(* IEC 61131-3 sources: RL_MAR/experiments/comparison/llm4plc/results/gpt-4o-mini_20260506_100619/20260506_101124, 4 files *)

(* ---- generated_code_iteration_0.st ---- *)
ructured-text
FUNCTION_BLOCK TruckGarage
VAR_INPUT
    enter_flag : BOOL;
    exit_flag : BOOL;
    VehicleNumber_in : INT;
END_VAR
VAR_OUTPUT
    truck : T_TRUCK_INFO;
END_VAR
VAR_IN_OUT
    garage : ARRAY[1..3, 1..5] OF T_GARAGE_SLOT;
END_VAR
VAR
    state : INT; // THE STATE VARIABLE
    row : INT; // THE CURRENT row being checked for parking
    col : INT; // THE CURRENT column being checked for parking
    found : BOOL; // Flag to indicate if a parking space has been found
    exit_row : INT; // Row of the vehicle to be exited
    exit_col : INT; // Column of the vehicle to be exited
    exit_found : BOOL; // Flag to indicate if the vehicle to be exited is found
END_VAR

// STATE MACHINE
IF state = 0 THEN // IDLE STATE
    IF enter_flag = TRUE AND exit_flag = FALSE THEN
        state := 1; // Transition to ALLOCATE PARKING SPACE
    ELSIF exit_flag = TRUE AND enter_flag = FALSE THEN
        state := 2; // Transition to RELEASE PARKING SPACE
    END_IF

ELSIF state = 1 THEN // ALLOCATE PARKING SPACE
    found := FALSE;
    FOR row := 3 TO 1 BY -1 DO
        FOR col := 5 TO 1 BY -1 DO
            IF garage[row, col].Occupied = FALSE THEN
                garage[row, col].Occupied := TRUE;
                garage[row, col].VehicleNumber := VehicleNumber_in;
                truck.row := row;
                truck.col := col;
                truck.VehicleNumber := VehicleNumber_in;
                found := TRUE;
                EXIT; // Exit the inner loop
            END_IF
        END_FOR
        IF found THEN
            EXIT; // Exit the outer loop
        END_IF
    END_FOR
    state := 0; // Transition back to IDLE STATE

ELSIF state = 2 THEN // RELEASE PARKING SPACE
    exit_found := FALSE;
    FOR row := 1 TO 3 DO
        FOR col := 1 TO 5 DO
            IF garage[row, col].VehicleNumber = VehicleNumber_in THEN
                garage[row, col].Occupied := FALSE;
                garage[row, col].VehicleNumber := 0; // Clear the VehicleNumber
                truck.row := row;
                truck.col := col;
                truck.VehicleNumber := VehicleNumber_in;
                exit_found := TRUE;
                EXIT; // Exit the inner loop
            END_IF
        END_FOR
        IF exit_found THEN
            EXIT; // Exit the outer loop
        END_IF
    END_FOR
    state := 0; // Transition back to IDLE STATE
END_IF

END_FUNCTION_BLOCK

(* ---- generated_code_iteration_1.st ---- *)
START_REASON
The errors occurred because the type 'T_TRUCK_INFO' is unknown in the context of the provided Structured Text (ST) code. This suggests that the type definition for 'T_TRUCK_INFO' has not been included or defined in the code. Additionally, the variable sections should be closed with "END_VAR" instead of "END_VAR_OUTPUT" or "END_VAR_INPUT". To resolve these issues, I will define the necessary types and ensure the variable sections are correctly closed.
END_REASON

START_ST
FUNCTION_BLOCK TruckGarage
VAR_INPUT
    enter_flag : BOOL;
    exit_flag : BOOL;
    VehicleNumber_in : INT;
END_VAR
VAR_OUTPUT
    truck : T_TRUCK_INFO;
END_VAR
VAR_IN_OUT
    garage : ARRAY[1..3, 1..5] OF T_GARAGE_SLOT;
END_VAR
VAR
    state : INT; // THE STATE VARIABLE
    row : INT; // THE CURRENT row being checked for parking
    col : INT; // THE CURRENT column being checked for parking
    found : BOOL; // Flag to indicate if a parking space has been found
    exit_row : INT; // Row of the vehicle to be exited
    exit_col : INT; // Column of the vehicle to be exited
    exit_found : BOOL; // Flag to indicate if the vehicle to be exited is found
END_VAR

// TYPE DEFINITIONS
TYPE T_TRUCK_INFO :
STRUCT
    row : INT;
    col : INT;
    VehicleNumber : INT;
END_STRUCT
END_TYPE

TYPE T_GARAGE_SLOT :
STRUCT
    Occupied : BOOL;
    VehicleNumber : INT;
END_STRUCT
END_TYPE

// STATE MACHINE
IF state = 0 THEN // IDLE STATE
    IF enter_flag = TRUE AND exit_flag = FALSE THEN
        state := 1; // Transition to ALLOCATE PARKING SPACE
    ELSIF exit_flag = TRUE AND enter_flag = FALSE THEN
        state := 2; // Transition to RELEASE PARKING SPACE
    END_IF

ELSIF state = 1 THEN // ALLOCATE PARKING SPACE
    found := FALSE;
    FOR row := 3 TO 1 BY -1 DO
        FOR col := 5 TO 1 BY -1 DO
            IF garage[row, col].Occupied = FALSE THEN
                garage[row, col].Occupied := TRUE;
                garage[row, col].VehicleNumber := VehicleNumber_in;
                truck.row := row;
                truck.col := col;
                truck.VehicleNumber := VehicleNumber_in;
                found := TRUE;
                EXIT; // Exit the inner loop
            END_IF
        END_FOR
        IF found THEN
            EXIT; // Exit the outer loop
        END_IF
    END_FOR
    state := 0; // Transition back to IDLE STATE

ELSIF state = 2 THEN // RELEASE PARKING SPACE
    exit_found := FALSE;
    FOR row := 1 TO 3 DO
        FOR col := 1 TO 5 DO
            IF garage[row, col].VehicleNumber = VehicleNumber_in THEN
                garage[row, col].Occupied := FALSE;
                garage[row, col].VehicleNumber := 0; // Clear the VehicleNumber
                truck.row := row;
                truck.col := col;
                truck.VehicleNumber := VehicleNumber_in;
                exit_found := TRUE;
                EXIT; // Exit the inner loop
            END_IF
        END_FOR
        IF exit_found THEN
            EXIT; // Exit the outer loop
        END_IF
    END_FOR
    state := 0; // Transition back to IDLE STATE
END_IF

END_FUNCTION_BLOCK
END_ST

(* ---- generated_code_iteration_2.st ---- *)
START_REASON
The errors occurred because the type 'T_TRUCK_INFO' was defined after it was used in the variable declarations. In Structured Text (ST), types must be defined before they are referenced. Additionally, the variable sections must be closed with "END_VAR" instead of "END_VAR_OUTPUT" or "END_VAR_INPUT". To resolve these issues, I will move the type definitions to the beginning of the code and ensure the variable sections are correctly closed.
END_REASON

START_ST
FUNCTION_BLOCK TruckGarage
// TYPE DEFINITIONS
TYPE T_TRUCK_INFO :
STRUCT
    row : INT;
    col : INT;
    VehicleNumber : INT;
END_STRUCT
END_TYPE

TYPE T_GARAGE_SLOT :
STRUCT
    Occupied : BOOL;
    VehicleNumber : INT;
END_STRUCT
END_TYPE

VAR_INPUT
    enter_flag : BOOL;
    exit_flag : BOOL;
    VehicleNumber_in : INT;
END_VAR
VAR_OUTPUT
    truck : T_TRUCK_INFO;
END_VAR
VAR_IN_OUT
    garage : ARRAY[1..3, 1..5] OF T_GARAGE_SLOT;
END_VAR
VAR
    state : INT; // THE STATE VARIABLE
    row : INT; // THE CURRENT row being checked for parking
    col : INT; // THE CURRENT column being checked for parking
    found : BOOL; // Flag to indicate if a parking space has been found
    exit_row : INT; // Row of the vehicle to be exited
    exit_col : INT; // Column of the vehicle to be exited
    exit_found : BOOL; // Flag to indicate if the vehicle to be exited is found
END_VAR

// STATE MACHINE
IF state = 0 THEN // IDLE STATE
    IF enter_flag = TRUE AND exit_flag = FALSE THEN
        state := 1; // Transition to ALLOCATE PARKING SPACE
    ELSIF exit_flag = TRUE AND enter_flag = FALSE THEN
        state := 2; // Transition to RELEASE PARKING SPACE
    END_IF

ELSIF state = 1 THEN // ALLOCATE PARKING SPACE
    found := FALSE;
    FOR row := 3 TO 1 BY -1 DO
        FOR col := 5 TO 1 BY -1 DO
            IF garage[row, col].Occupied = FALSE THEN
                garage[row, col].Occupied := TRUE;
                garage[row, col].VehicleNumber := VehicleNumber_in;
                truck.row := row;
                truck.col := col;
                truck.VehicleNumber := VehicleNumber_in;
                found := TRUE;
                EXIT; // Exit the inner loop
            END_IF
        END_FOR
        IF found THEN
            EXIT; // Exit the outer loop
        END_IF
    END_FOR
    state := 0; // Transition back to IDLE STATE

ELSIF state = 2 THEN // RELEASE PARKING SPACE
    exit_found := FALSE;
    FOR row := 1 TO 3 DO
        FOR col := 1 TO 5 DO
            IF garage[row, col].VehicleNumber = VehicleNumber_in THEN
                garage[row, col].Occupied := FALSE;
                garage[row, col].VehicleNumber := 0; // Clear the VehicleNumber
                truck.row := row;
                truck.col := col;
                truck.VehicleNumber := VehicleNumber_in;
                exit_found := TRUE;
                EXIT; // Exit the inner loop
            END_IF
        END_FOR
        IF exit_found THEN
            EXIT; // Exit the outer loop
        END_IF
    END_FOR
    state := 0; // Transition back to IDLE STATE
END_IF

END_FUNCTION_BLOCK
END_ST

(* ---- generated_code_iteration_3.st ---- *)
START_REASON
The errors occurred because the variable sections must be defined using "VAR", "VAR_INPUT", "VAR_OUTPUT", or "VAR_IN_OUT" correctly. The type definitions were placed correctly, but the variable declarations were not structured properly according to the feedback. I will ensure that the variable sections are defined correctly and close them with "END_VAR".
END_REASON

START_ST
FUNCTION_BLOCK TruckGarage
// TYPE DEFINITIONS
TYPE T_TRUCK_INFO :
STRUCT
    row : INT;
    col : INT;
    VehicleNumber : INT;
END_STRUCT
END_TYPE

TYPE T_GARAGE_SLOT :
STRUCT
    Occupied : BOOL;
    VehicleNumber : INT;
END_STRUCT
END_TYPE

VAR_INPUT
    enter_flag : BOOL;
    exit_flag : BOOL;
    VehicleNumber_in : INT;
END_VAR

VAR_OUTPUT
    truck : T_TRUCK_INFO;
END_VAR

VAR_IN_OUT
    garage : ARRAY[1..3, 1..5] OF T_GARAGE_SLOT;
END_VAR

VAR
    state : INT; // THE STATE VARIABLE
    row : INT; // THE CURRENT row being checked for parking
    col : INT; // THE CURRENT column being checked for parking
    found : BOOL; // Flag to indicate if a parking space has been found
    exit_row : INT; // Row of the vehicle to be exited
    exit_col : INT; // Column of the vehicle to be exited
    exit_found : BOOL; // Flag to indicate if the vehicle to be exited is found
END_VAR

// STATE MACHINE
IF state = 0 THEN // IDLE STATE
    IF enter_flag = TRUE AND exit_flag = FALSE THEN
        state := 1; // Transition to ALLOCATE PARKING SPACE
    ELSIF exit_flag = TRUE AND enter_flag = FALSE THEN
        state := 2; // Transition to RELEASE PARKING SPACE
    END_IF

ELSIF state = 1 THEN // ALLOCATE PARKING SPACE
    found := FALSE;
    FOR row := 3 TO 1 BY -1 DO
        FOR col := 5 TO 1 BY -1 DO
            IF garage[row, col].Occupied = FALSE THEN
                garage[row, col].Occupied := TRUE;
                garage[row, col].VehicleNumber := VehicleNumber_in;
                truck.row := row;
                truck.col := col;
                truck.VehicleNumber := VehicleNumber_in;
                found := TRUE;
                EXIT; // Exit the inner loop
            END_IF
        END_FOR
        IF found THEN
            EXIT; // Exit the outer loop
        END_IF
    END_FOR
    state := 0; // Transition back to IDLE STATE

ELSIF state = 2 THEN // RELEASE PARKING SPACE
    exit_found := FALSE;
    FOR row := 1 TO 3 DO
        FOR col := 1 TO 5 DO
            IF garage[row, col].VehicleNumber = VehicleNumber_in THEN
                garage[row, col].Occupied := FALSE;
                garage[row, col].VehicleNumber := 0; // Clear the VehicleNumber
                truck.row := row;
                truck.col := col;
                truck.VehicleNumber := VehicleNumber_in;
                exit_found := TRUE;
                EXIT; // Exit the inner loop
            END_IF
        END_FOR
        IF exit_found THEN
            EXIT; // Exit the outer loop
        END_IF
    END_FOR
    state := 0; // Transition back to IDLE STATE
END_IF

END_FUNCTION_BLOCK
END_ST
